(* CODESYS project 2 Mixer Process .project

Project tree, tasks and I/O mapping:
  Device : CODESYS Control Win V3, 3S - Smart Software Solutions GmbH, order no. 305021, version 3.5.7.0
    application Application
      libraries: Standard, * (System)
      task MainTask (cyclic, interval t#20ms, priority 1) calls PLC_PRG
      task VISU_TASK (cyclic, interval 100 ms, priority 31) calls VisuElems.Visu_Prg
      program PLC_PRG [LD]
      visualisation Visualization
  text list GlobalTextList
*)

// Device/Application/PLC_PRG
PROGRAM PLC_PRG
VAR
	TON_01: TON;
	TP_02: TP;
	TON_02: TON;
	start: BOOL;
	stop: BOOL;
	cycle_off: BOOL;
	cycle_on: BOOL;
	level_5: BOOL;
	outlet_valve1: BOOL;
	level_a: BOOL;
	lls: BOOL;
	inlet_valve1: BOOL;
	inlet_valve2: BOOL;
	temp_sensor: BOOL;
	level_b: BOOL;
	heater: BOOL;
	output: BOOL;
	agitator_motor: BOOL;
	T: TIME;
	TT: TIME;
	TTTT: TIME;
END_VAR

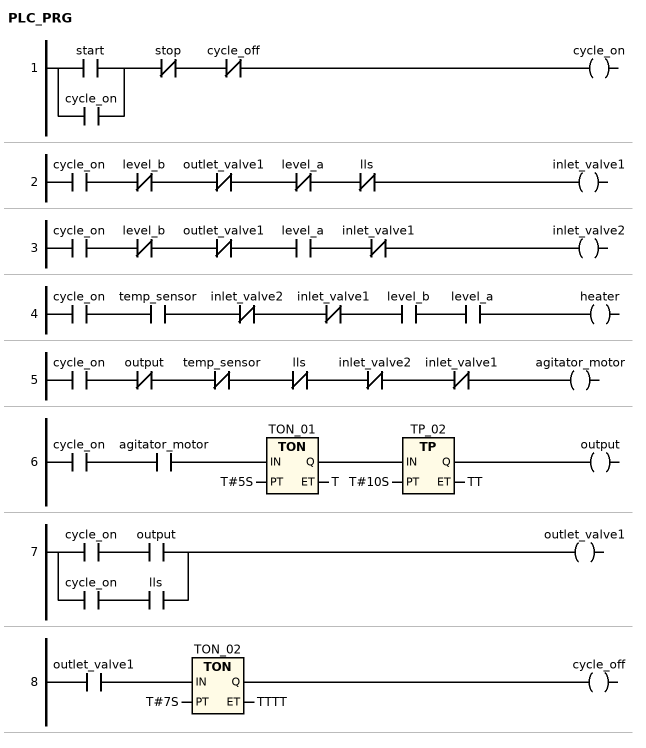
// NETWORK 1
cycle_on := (start OR cycle_on) AND NOT stop AND NOT cycle_off;

// NETWORK 2
inlet_valve1 := cycle_on AND NOT level_b AND NOT outlet_valve1 AND NOT level_a AND NOT lls;

// NETWORK 3
inlet_valve2 := cycle_on AND NOT level_b AND NOT outlet_valve1 AND level_a AND NOT inlet_valve1;

// NETWORK 4
heater := cycle_on AND temp_sensor AND NOT inlet_valve2 AND NOT inlet_valve1 AND level_b AND level_a;

// NETWORK 5
agitator_motor := cycle_on AND NOT output AND NOT temp_sensor AND NOT lls AND NOT inlet_valve2 AND NOT inlet_valve1;

// NETWORK 6
TON_01(IN := cycle_on AND agitator_motor, PT := T#5S, ET => T); // TON
TP_02(IN := TON_01.Q, PT := T#10S, ET => TT); // TP
output := TP_02.Q;

// NETWORK 7
outlet_valve1 := cycle_on AND output OR cycle_on AND lls;

// NETWORK 8
TON_02(IN := outlet_valve1, PT := T#7S, ET => TTTT); // TON
cycle_off := TON_02.Q;

END_PROGRAM

// Device/Application/Visualization
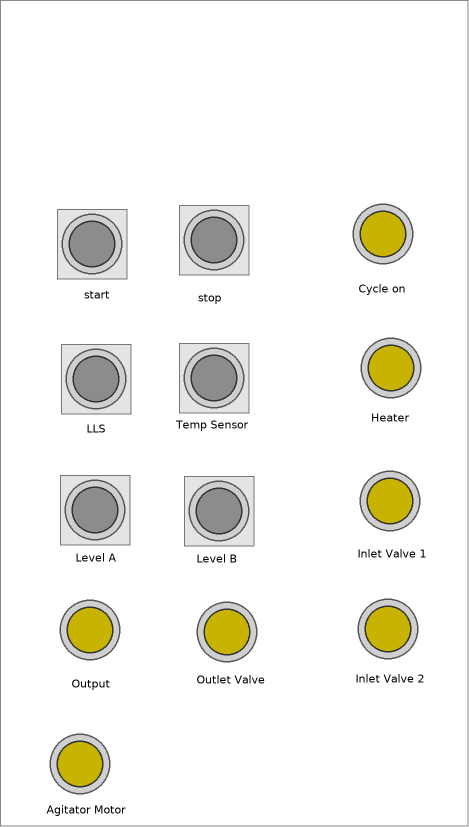
VISUALIZATION Visualization  // 469x827
    PushSwitchLed (57,209 70x70), variable: PLC_PRG.start, behaviour: TOGGLE, style: Switch-PushSwitchLed-Gray
    PushSwitchLed (184,476 70x70), variable: PLC_PRG.level_b, behaviour: TOGGLE, style: Switch-PushSwitchLed-Gray
    PushSwitchLed (179,343 70x70), variable: PLC_PRG.temp_sensor, behaviour: TOGGLE, style: Switch-PushSwitchLed-Gray
    PushSwitchLed (179,205 70x70), variable: PLC_PRG.stop, behaviour: TOGGLE, style: Switch-PushSwitchLed-Gray
    PushSwitchLed (61,344 70x70), variable: PLC_PRG.lls, behaviour: TOGGLE, style: Switch-PushSwitchLed-Gray
    PushSwitchLed (60,475 70x70), variable: PLC_PRG.level_a, behaviour: TOGGLE, style: Switch-PushSwitchLed-Gray
    Lamp1 (348,199 70x70), variable: PLC_PRG.cycle_on, style: Lamp-Lamp1-Yellow
    Lamp1 (45,729 70x70), variable: PLC_PRG.agitator_motor, style: Lamp-Lamp1-Yellow
    Lamp1 (353,594 70x70), variable: PLC_PRG.inlet_valve2, style: Lamp-Lamp1-Yellow
    Lamp1 (355,466 70x70), variable: PLC_PRG.inlet_valve1, style: Lamp-Lamp1-Yellow
    Lamp1 (356,333 70x70), variable: PLC_PRG.heater, style: Lamp-Lamp1-Yellow
    Lamp1 (192,597 70x70), variable: PLC_PRG.outlet_valve1, style: Lamp-Lamp1-Yellow
    Lamp1 (55,595 70x70), variable: PLC_PRG.output, style: Lamp-Lamp1-Yellow
    Label (22,280 150x30), "start"
    Label (135,283 150x30), "stop"
    Label (21,414 150x30), "LLS"
    Label (137,410 150x30), "Temp Sensor"
    Label (21,543 150x30), "Level A"
    Label (142,544 150x30), "Level B"
    Label (16,669 150x30), "Output"
    Label (156,665 150x30), "Outlet Valve"
    Label (307,274 150x30), "Cycle on"
    Label (315,403 150x30), "Heater"
    Label (317,539 150x30), "Inlet Valve 1"
    Label (315,664 150x30), "Inlet Valve 2"
    Label (11,795 150x30), "Agitator Motor"
END_VISUALIZATION
